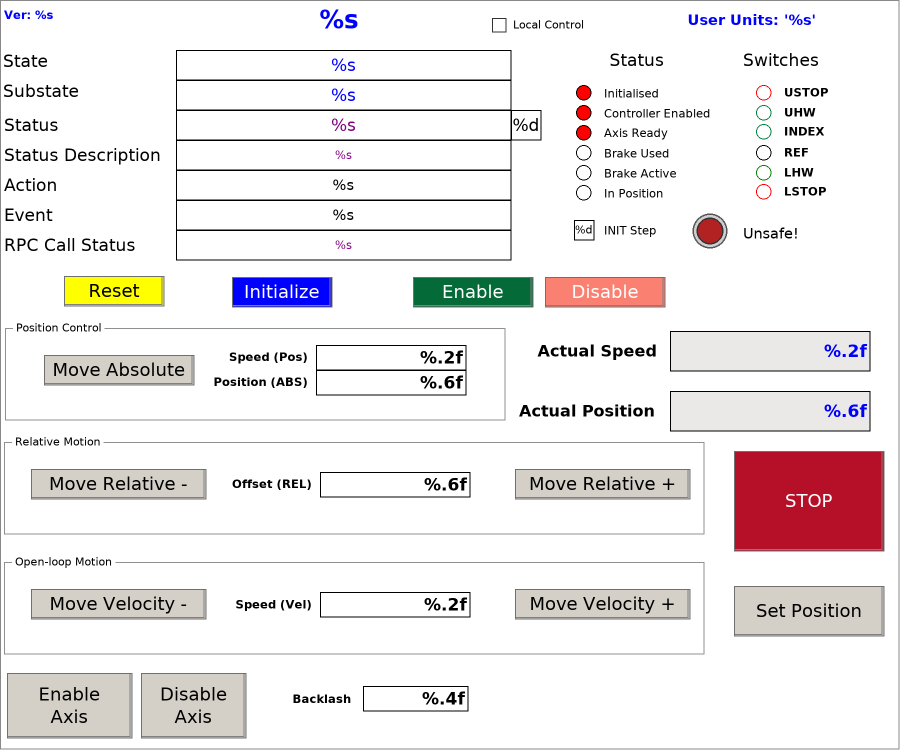
VISUALIZATION GUI_TEMPLATE_NOTT_MOTOR_CONTROL  // 900x750
VAR_IN_OUT
	m_Instance:	FB_NOTT_MOTOR;
END_VAR
VAR
	m_lrOffSet : LREAL := 0;
END_VAR
    GroupBox (4,554 700x100), "Open-loop Motion"
        Button (511,35 175x30), "Move Velocity +", input disabled if: NOT m_Instance.stat.bLocal OR NOT m_Instance.in_bSafe
            OnMouseDown: execute {
                m_Instance.ctrl.bLocalCmd := TRUE;
                m_Instance.ctrl.nCommand := E_MOTOR_COMMAND.MOTOR_MOVE;
                m_Instance.ctrl.nMoveType := E_MOTOR_MOVE_TYPE.VELOCITY;
                m_Instance.ctrl.nDirection := MC_Positive_Direction;
                m_Instance.ctrl.bExecute := TRUE;
            }
    GroupBox (4,434 700x100), "Relative Motion"
    GroupBox (5,320 500x100), "Position Control"
    Rectangle (176,50 335x30), "%s", text variable: m_Instance.stat.sState
    Rectangle (176,80 335x30), "%s", text variable: m_Instance.stat.sSubstate
    Button (64,276 100x30), "Reset", input disabled if: NOT m_Instance.stat.bLocal OR NOT m_Instance.in_bSafe
        OnMouseDown: execute {
            m_Instance.ctrl.bLocalCmd := TRUE;
            m_Instance.ctrl.nCommand := E_MOTOR_COMMAND.RESET;
            m_Instance.ctrl.bExecute := TRUE;
        }
    Button (232,277 100x30), "Initialize", input disabled if: NOT m_Instance.stat.bLocal OR NOT m_Instance.in_bSafe
        OnMouseDown: execute {
            m_Instance.ctrl.bLocalCmd := TRUE;
            m_Instance.ctrl.nCommand := E_MOTOR_COMMAND.INIT;
            m_Instance.ctrl.bExecute := TRUE;
        }
    Button (734,451 150x100), "STOP", input disabled if: NOT m_Instance.stat.bLocal OR NOT m_Instance.in_bSafe
        OnMouseDown: execute {
            m_Instance.ctrl.bLocalCmd := TRUE;
            m_Instance.ctrl.nCommand := E_MOTOR_COMMAND.STOP;
            m_Instance.ctrl.bExecute := TRUE;
        }
    Button (413,277 120x30), "Enable", input disabled if: NOT m_Instance.stat.bLocal OR NOT m_Instance.in_bSafe
        OnMouseDown: execute {
            m_Instance.ctrl.bLocalCmd := TRUE;
            m_Instance.ctrl.nCommand := E_MOTOR_COMMAND.ENABLE;
            m_Instance.ctrl.bExecute := TRUE;
        }
    Button (545,277 120x30), "Disable", input disabled if: NOT m_Instance.stat.bLocal OR NOT m_Instance.in_bSafe
        OnMouseDown: execute {
            m_Instance.ctrl.bLocalCmd := TRUE;
            m_Instance.ctrl.nCommand := E_MOTOR_COMMAND.DISABLE;
            m_Instance.ctrl.bExecute := TRUE;
        }
    Rectangle (0,46 170x30), "State"
    Rectangle (0,76 170x30), "Substate"
    Rectangle (176,110 335x30), "%s", text variable: m_Instance.stat.sStatus
    Rectangle (176,140 335x30), "%s", tooltip "Additional information mostly used for description of errors", text variable: m_Instance.stat.sErrorText
    Rectangle (1,110 170x30), "Status"
    Rectangle (1,140 170x30), "Status Description"
    Rectangle (176,170 335x30), "%s", text variable: m_Instance.stat.sActionDesc
    Rectangle (176,200 335x30), "%s", text variable: m_Instance.stat.sEventDesc
    Rectangle (1,170 170x30), "Action"
    Rectangle (1,200 170x30), "Event"
    Rectangle (223,2 232x35), "%s", text variable: m_Instance.sName
    Checkbox (490,10 116x30), "Local Control", variable: m_Instance.stat.bLocal
    Rectangle (591,45 92x30), "Status"
    Rectangle (511,110 30x30), "%d", text variable: m_Instance.stat.nStatus
    Rectangle (735,45 92x30), "Switches"
    Button (734,586 150x50), "Set Position", input disabled if: NOT m_Instance.stat.bLocal OR NOT m_Instance.in_bSafe
        OnMouseDown: execute {
            m_Instance.ctrl.bLocalCmd := TRUE;
            m_Instance.ctrl.nCommand := E_MOTOR_COMMAND.SET_POSITION;
            m_Instance.ctrl.bExecute := TRUE;
        }
    Rectangle (781,85 50x15), "USTOP"
    Ellipse (756,85 15x15), colour toggle: m_Instance.stat.signals[5].bActive
    Ellipse (756,105 15x15), colour toggle: m_Instance.stat.signals[4].bActive
    Ellipse (756,165 15x15), colour toggle: m_Instance.stat.signals[1].bActive
    Ellipse (756,184 15x15), colour toggle: m_Instance.stat.signals[0].bActive
    Ellipse (756,145 15x15), colour toggle: m_Instance.stat.signals[2].bActive
    Rectangle (781,124 50x15), "INDEX"
    Rectangle (781,105 50x15), "UHW"
    Rectangle (781,145 50x15), "REF"
    Rectangle (781,165 50x15), "LHW"
    Rectangle (781,184 50x15), "LSTOP"
    Ellipse (756,124 15x15), colour toggle: m_Instance.stat.signals[3].bActive
    Group (259,686 209x25)
        Rectangle (0,3 95x20), "Backlash"
        Rectangle (104,0 105x25), "%.4f", text variable: m_Instance.cfg.lrBacklash
            OnMouseDown: write the text variable via Default
    Button (44,355 150x30), "Move Absolute", input disabled if: NOT m_Instance.stat.bLocal OR NOT m_Instance.in_bSafe
        OnMouseDown: execute {
            m_Instance.ctrl.bLocalCmd := TRUE;
            m_Instance.ctrl.lrVelocity:=(m_Instance.cfg.lrDefaultVelocity);
            m_Instance.ctrl.nCommand := E_MOTOR_COMMAND.MOTOR_MOVE;
            m_Instance.ctrl.nMoveType := E_MOTOR_MOVE_TYPE.ABSOLUTE;
            m_Instance.ctrl.bExecute := TRUE;
        }
    Group (216,370 250x25)
        Rectangle (0,2 95x20), "Position (ABS)"
        Rectangle (100,0 150x25), "%.6f", tooltip "Absolute position used by "MOVE ABS"", text variable: m_Instance.ctrl.lrPosition
            OnMouseDown: write the text variable via Default
    Group (216,345 250x25)
        Rectangle (0,2 95x20), "Speed (Pos)"
        Rectangle (100,0 150x25), "%.2f", text variable: m_Instance.cfg.lrDefaultVelocity
            OnMouseDown: write the text variable via Default
    Rectangle (601,161 90x25), "Brake Active"
    Ellipse (576,165 15x15), tooltip "RED = Applied BLANK = Released", colour toggle: (m_Instance.stat.bBrakeActive) <> 0
    Ellipse (576,85 15x15), tooltip "GREEN = Initialised RED = Not Initialised", text variable: m_Instance.stat.bInitialised, colour toggle: m_Instance.stat.bInitialised
    Rectangle (601,81 90x25), "Initialised"
    Rectangle (601,101 125x25), "Controller Enabled"
    Rectangle (601,121 90x24), "Axis Ready"
    Rectangle (601,141 90x25), "Brake Used"
    Ellipse (576,105 15x15), tooltip "GREEN = Enabled RED = Disabled", colour toggle: m_Instance.stat.bEnabled
    Ellipse (576,125 15x15), tooltip "GREEN = Ready RED = Not Ready", colour toggle: m_Instance.stat.bAxisReady
    Ellipse (576,145 15x15), tooltip "BLUE = Used BLANK = Not Used", colour toggle: m_Instance.cfg.bUseBrake
    Rectangle (574,220 20x20), "%d", text variable: m_Instance.stat.nInitStep
    Rectangle (601,218 90x25), "INIT Step"
    Rectangle (1,230 170x30), "RPC Call Status"
    Rectangle (176,230 335x30), "%s", text variable: m_Instance.stat.sRPCErrorText
    Rectangle (601,181 90x25), "In Position"
    Ellipse (576,185 15x15), tooltip "GREEN = In Position BLANK = Not In Position (or not used)", colour toggle: (m_Instance.stat.bInPosition) <> 0
    Button (7,673 125x65), "Enable Axis", input disabled if: NOT m_Instance.stat.bLocal OR NOT m_Instance.in_bSafe
        OnMouseDown: execute { m_Instance.stat.bEnabled := TRUE; }
    Button (141,673 105x65), "Disable Axis", input disabled if: NOT m_Instance.stat.bLocal OR NOT m_Instance.in_bSafe
        OnMouseDown: execute { m_Instance.stat.bEnabled := FALSE; }
    Rectangle (616,5 203x30), "User Units: '%s'", text variable: m_Instance.stat.axis.sUnits
    Rectangle (1,0 99x30), "Ver: %s", tooltip "'Motor.library version'", text variable: m_Instance.stat.sLibVersion, input disabled if: true
    Lamp1 (690,211 40x40), tooltip "If active, it is not safe to operate the motor.", variable: NOT m_Instance.in_bSafe, invisible if: m_Instance.in_bSafe, style: Lamp-Lamp1-Red
    Rectangle (730,223 82x21), "Unsafe!", invisible if: m_Instance.in_bSafe
    Group (510,331 360x40)
        Rectangle (160,0 200x40), "%.2f", text variable: m_Instance.stat.lrVelActual, input disabled if: false
        Rectangle (0,5 150x30), "Actual Speed"
    Group (508,391 362x40)
        Rectangle (162,0 200x40), "%.6f", text variable: m_Instance.stat.lrPosActual, input disabled if: false
        Rectangle (0,5 150x30), "Actual Position"
    Group (220,592 250x25)
        Rectangle (0,0 95x25), "Speed (Vel)"
        Rectangle (100,0 150x25), "%.2f", text variable: m_Instance.ctrl.lrVelocity
            OnMouseDown: write the text variable via Default
    Button (31,589 175x30), "Move Velocity -", input disabled if: NOT m_Instance.stat.bLocal OR NOT m_Instance.in_bSafe
        OnMouseDown: execute {
            m_Instance.ctrl.bLocalCmd := TRUE;
            m_Instance.ctrl.nCommand := E_MOTOR_COMMAND.MOTOR_MOVE;
            m_Instance.ctrl.nMoveType := E_MOTOR_MOVE_TYPE.VELOCITY;
            m_Instance.ctrl.nDirection := MC_Negative_Direction;
            m_Instance.ctrl.bExecute := TRUE;
        }
    Button (31,469 175x30), "Move Relative -", input disabled if: NOT m_Instance.stat.bLocal OR NOT m_Instance.in_bSafe
        OnMouseDown: execute {
            m_Instance.ctrl.bLocalCmd := TRUE;
            m_Instance.ctrl.lrOffset := m_lrOffSet * (-1);
            m_Instance.ctrl.lrVelocity:=(m_Instance.cfg.lrDefaultVelocity);
            m_Instance.ctrl.nCommand := E_MOTOR_COMMAND.MOTOR_MOVE;
            m_Instance.ctrl.nMoveType := E_MOTOR_MOVE_TYPE.RELATIVE;
            m_Instance.ctrl.bExecute := TRUE;
        }
    Group (220,472 250x25)
        Rectangle (0,2 95x20), "Offset (REL)"
        Rectangle (100,0 150x25), "%.6f", tooltip "Relative offset used by "MOVE REL"", text variable: m_lrOffSet
            OnMouseDown: write the text variable via Default
    Button (515,469 175x30), "Move Relative +", input disabled if: NOT m_Instance.stat.bLocal OR NOT m_Instance.in_bSafe
        OnMouseDown: execute {
            m_Instance.ctrl.bLocalCmd := TRUE;
            m_Instance.ctrl.lrOffset := m_lrOffSet;
            m_Instance.ctrl.lrVelocity:=(m_Instance.cfg.lrDefaultVelocity);
            m_Instance.ctrl.nCommand := E_MOTOR_COMMAND.MOTOR_MOVE;
            m_Instance.ctrl.nMoveType := E_MOTOR_MOVE_TYPE.RELATIVE;
            m_Instance.ctrl.bExecute := TRUE;
        }
END_VISUALIZATION

(* stored: Version 1.1.0.1, ProductVersion 3.1.4024.14
   Visu GUI_TEMPLATE_NOTT_MOTOR_CONTROL: Id {208abcb1-f1a3-4a00-92a5-f362cd7556ac} *)
